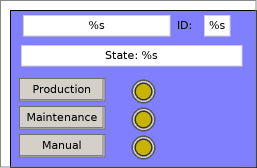
VISUALIZATION V_Module  // 257x168
VAR_IN_OUT
	stVisu				: ST_PMLModuleBaseVISU;
END_VAR
    RoundedRectangle (10,10 247x158)
    Textfield (23,15 147x21), "%s", text variable: stVisu.sModuleName
    Textfield (204,15 26x21), "%s", text variable: stVisu.nModuleID
    Label (165,14 39x23), "ID:"
    Textfield (21,45 221x21), "State: %s", text variable: stVisu.eState
    Button (19,78 86x23), "Production"
        tap stVisu.bProductionPressed
    Button (19,106 86x23), "Maintenance"
        tap stVisu.bMaintenancePressed
    Button (19,134 86x23), "Manual"
        tap stVisu.bManualPressed
    Lamp1 (130,78 27x27), variable: stVisu.eMode = E_PMLProtectedUnitMode.ePMLProtUnitMode_Production, style: Lamp-Lamp1-Yellow
    Lamp1 (130,106 27x27), variable: stVisu.eMode = E_PMLProtectedUnitMode.ePMLProtUnitMode_Maintenance, style: Lamp-Lamp1-Yellow
    Lamp1 (130,134 27x27), variable: stVisu.eMode = E_PMLProtectedUnitMode.ePMLProtUnitMode_Manual, style: Lamp-Lamp1-Yellow
END_VISUALIZATION

(* stored: Version 1.1.0.1, ProductVersion 3.1.4024.10
   Visu V_Module: Id {ab5ca517-81c1-49dd-92aa-b6c97677d45a} *)
